FUNCTION_BLOCK OutputChannelAdptd (* Composite Function Block Type *)
  (* Standard: 61499-2 *)
  (* Version 0.0, 09/10/2018, Atmojo, nxtControl GmbH, template *)
  PACKAGE Main;
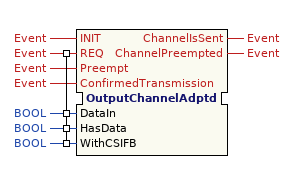
  EVENT_INPUT
    INIT;
    REQ WITH DataIn, HasData, WithCSIFB; (* Normal Execution Request *)
    Preempt;
    ConfirmedTransmission;
  END_EVENT
  EVENT_OUTPUT
    ChannelIsSent; (* Initialization Confirm *)
    ChannelPreempted; (* Execution Confirmation *)
  END_EVENT
  VAR_INPUT
    DataIn : BOOL;
    HasData : BOOL;
    WithCSIFB : BOOL;
  END_VAR
END_FUNCTION_BLOCK
